TYPE T_String : STRING; END_TYPE

(* stored: Version 1.1.0.1, ProductVersion 3.1.4024.4
   DUT T_String: Id {ecdf3a42-0023-41ec-9520-a8f3827576b5} *)
